TYPE E_LampState : 
(
	Off := 0,
    Steady := 1,
    FastFlash := 2,
    SlowFlash := 4
);
END_TYPE

(* stored: Version 1.1.0.1, ProductVersion 3.1.0.36
   DUT E_LampState: Id {75b52d8c-08bb-42cc-9dc1-f3d5a3a90936} *)
